FUNCTION NowDT : DT
VAR_INPUT
END_VAR
VAR
	timeAsFileTime: T_FILETIME;
END_VAR
VAR_STAT
	fbSystemTime: GETSYSTEMTIME;
END_VAR

fbSystemTime(
	timeLoDW =>timeAsFileTime.dwLowDateTime,
	timeHiDW =>timeAsFileTime.dwHighDateTime 
);
NowDT := FILETIME_TO_DT( timeAsFileTime );

END_FUNCTION

(* stored: Version 1.1.0.1, ProductVersion 3.1.4024.6
   POU NowDT: Id {40f516c8-c703-4526-8fc3-882dac645da7}, SpecialFunc None *)
